{attribute 'qualified_only'}
// CoE entry in the dictionary, includes index and the subindex
TYPE ST_CoeEntry :
STRUCT
	Index		: WORD;
	Subindex	: BYTE;
END_STRUCT
END_TYPE

(* stored: Version 1.1.0.1, ProductVersion 3.1.4024.14
   DUT ST_CoeEntry: Id {f015f297-00e6-0477-1aab-3c2a88aa8019} *)
